LIN {X 0,Y 86.241,Z 1157.577,A -85,B 0,C 180,E1 5429.612,E2 5429.612} C_VEL
LIN {X 0,Y 83.784,Z 1172.301,A -85,B 0,C 180,E1 5420.249,E2 5420.249} C_VEL
LIN {X 0,Y 83.269,Z 1185.193,A -85,B 0,C 180,E1 5410.109,E2 5410.109} C_VEL
LIN {X 0,Y 85.244,Z 1197.586,A -85,B 0,C 180,E1 5398.656,E2 5398.656} C_VEL
LIN {X 0,Y 91.359,Z 1209.722,A -85,B 0,C 180,E1 5386.067,E2 5386.067} C_VEL
LIN {X 0,Y 101.878,Z 1220.023,A -85,B 0,C 180,E1 5375.037,E2 5375.037} C_VEL
LIN {X 0,Y 114.698,Z 1227.862,A -85,B 0,C 180,E1 5366.799,E2 5366.799} C_VEL
LIN {X 0,Y 97.634,Z 1225.464,A -85,B 0,C 180,E1 5353.315,E2 5353.315} C_VEL
LIN {X 0,Y 88.981,Z 1221.588,A -85,B 0,C 180,E1 5336.7,E2 5336.7} C_VEL
LIN {X 0,Y 88.107,Z 1220.31,A -85,B 0,C 180,E1 5331.809,E2 5331.809} C_VEL
LIN {X 0,Y 85.061,Z 1227.697,A -85,B 0,C 180,E1 5324.282,E2 5324.282} C_VEL
LIN {X 0,Y 85.385,Z 1239.016,A -85,B 0,C 180,E1 5311.333,E2 5311.333} C_VEL
LIN {X 0,Y 86.182,Z 1243.374,A -85,B 0,C 180,E1 5305.333,E2 5305.333} C_VEL
LIN {X 0,Y 85.817,Z 1248.62,A -85,B 0,C 180,E1 5294.447,E2 5294.447} C_VEL
LIN {X 0,Y 90.743,Z 1255.131,A -85,B 0,C 180,E1 5277.312,E2 5277.312} C_VEL
LIN {X 0,Y 102.644,Z 1259.967,A -85,B 0,C 180,E1 5263.088,E2 5263.088} C_VEL
LIN {X 0,Y 89.773,Z 1251.394,A -85,B 0,C 180,E1 5248.616,E2 5248.616} C_VEL
LIN {X 0,Y 84.154,Z 1242.377,A -85,B 0,C 180,E1 5233.747,E2 5233.747} C_VEL
LIN {X 0,Y 82.846,Z 1235.817,A -85,B 0,C 180,E1 5224.153,E2 5224.153} C_VEL
LIN {X 0,Y 82.358,Z 1227.952,A -85,B 0,C 180,E1 5214.426,E2 5214.426} C_VEL
LIN {X 0,Y 83.548,Z 1216.638,A -85,B 0,C 180,E1 5202.591,E2 5202.591} C_VEL
LIN {X 0,Y 87.163,Z 1203.687,A -85,B 0,C 180,E1 5191.683,E2 5191.683} C_VEL
LIN {X 0,Y 88.042,Z 1198.552,A -85,B 0,C 180,E1 5187.954,E2 5187.954} C_VEL
LIN {X 0,Y 88.162,Z 1183.445,A -85,B 0,C 180,E1 5178.16,E2 5178.16} C_VEL
LIN {X 0,Y 89.756,Z 1178.502,A -85,B 0,C 180,E1 5175.416,E2 5175.416} C_VEL
LIN {X 0,Y 98.668,Z 1160.656,A -85,B 0,C 180,E1 5167.456,E2 5167.456} C_VEL
LIN {X 0,Y 108.892,Z 1140.068,A -85,B 0,C 180,E1 5160.845,E2 5160.845} C_VEL
LIN {X 0,Y 119.307,Z 1117.626,A -85,B 0,C 180,E1 5155.718,E2 5155.718} C_VEL
LIN {X 0,Y 129.224,Z 1093.9,A -85,B 0,C 180,E1 5151.794,E2 5151.794} C_VEL
LIN {X 0,Y 137.935,Z 1070.062,A -85,B 0,C 180,E1 5148.915,E2 5148.915} C_VEL
LIN {X 0,Y 145.83,Z 1044.502,A -85,B 0,C 180,E1 5146.657,E2 5146.657} C_VEL
LIN {X 0,Y 152.519,Z 1017.799,A -85,B 0,C 180,E1 5144.946,E2 5144.946} C_VEL
LIN {X 0,Y 182.121,Z 883.493,A -85,B 0,C 180,E1 5138.791,E2 5138.791} C_VEL
LIN {X 0,Y 178.666,Z 874.642,A -85,B 0,C 180,E1 5136.269,E2 5136.269} C_VEL
LIN {X 0,Y 168.951,Z 876.076,A -85,B 0,C 180,E1 5132.04,E2 5132.04} C_VEL
LIN {X 0,Y 161.363,Z 878.264,A -85,B 0,C 180,E1 5128.389,E2 5128.389} C_VEL
LIN {X 0,Y 158.218,Z 879.25,A -85,B 0,C 180,E1 5126.744,E2 5126.744} C_VEL
LIN {X 0,Y 157.864,Z 879.467,A -85,B 0,C 180,E1 5126.374,E2 5126.374} C_VEL
LIN {X 0,Y 158.802,Z 887.342,A -85,B 0,C 180,E1 5122.407,E2 5122.407} C_VEL
LIN {X 0,Y 137.912,Z 929.195,A -85,B 0,C 180,E1 5115.445,E2 5115.445} C_VEL
LIN {X 0,Y 129.417,Z 947.663,A -85,B 0,C 180,E1 5111.944,E2 5111.944} C_VEL
LIN {X 0,Y 118.078,Z 998.542,A -85,B 0,C 180,E1 5108.011,E2 5108.011} C_VEL
LIN {X 0,Y 108.514,Z 1037.175,A -85,B 0,C 180,E1 5103.701,E2 5103.701} C_VEL
LIN {X 0,Y 99.397,Z 1074.485,A -85,B 0,C 180,E1 5097.673,E2 5097.673} C_VEL
LIN {X 0,Y 91.918,Z 1104.757,A -85,B 0,C 180,E1 5091.009,E2 5091.009} C_VEL
LIN {X 0,Y 86.721,Z 1124.357,A -85,B 0,C 180,E1 5085.162,E2 5085.162} C_VEL
LIN {X 0,Y 82.161,Z 1140.976,A -85,B 0,C 180,E1 5078.365,E2 5078.365} C_VEL
LIN {X 0,Y 78.202,Z 1157.109,A -85,B 0,C 180,E1 5069.627,E2 5069.627} C_VEL
LIN {X 0,Y 75.851,Z 1171.444,A -85,B 0,C 180,E1 5059.643,E2 5059.643} C_VEL
LIN {X 0,Y 75.568,Z 1184.592,A -85,B 0,C 180,E1 5048.369,E2 5048.369} C_VEL
LIN {X 0,Y 77.98,Z 1196.619,A -85,B 0,C 180,E1 5036.324,E2 5036.324} C_VEL
LIN {X 0,Y 84.068,Z 1207.905,A -85,B 0,C 180,E1 5024.124,E2 5024.124} C_VEL
LIN {X 0,Y 95.246,Z 1218.728,A -85,B 0,C 180,E1 5012.49,E2 5012.49} C_VEL
LIN {X 0,Y 104.27,Z 1224.54,A -85,B 0,C 180,E1 5006.526,E2 5006.526} C_VEL
LIN {X 0,Y 87.98,Z 1221.298,A -85,B 0,C 180,E1 4991.224,E2 4991.224} C_VEL
LIN {X 0,Y 81.108,Z 1216.92,A -85,B 0,C 180,E1 4973.223,E2 4973.223} C_VEL
LIN {X 0,Y 77.596,Z 1224.563,A -85,B 0,C 180,E1 4964.885,E2 4964.885} C_VEL
LIN {X 0,Y 77.861,Z 1236.114,A -85,B 0,C 180,E1 4950.726,E2 4950.726} C_VEL
LIN {X 0,Y 78.846,Z 1240.177,A -85,B 0,C 180,E1 4944.897,E2 4944.897} C_VEL
LIN {X 0,Y 78.56,Z 1244.991,A -85,B 0,C 180,E1 4934.487,E2 4934.487} C_VEL
LIN {X 0,Y 82.705,Z 1251.194,A -85,B 0,C 180,E1 4917.852,E2 4917.852} C_VEL
LIN {X 0,Y 93.414,Z 1256.211,A -85,B 0,C 180,E1 4903.24,E2 4903.24} C_VEL
LIN {X 0,Y 81.625,Z 1247.63,A -85,B 0,C 180,E1 4888.538,E2 4888.538} C_VEL
LIN {X 0,Y 76.334,Z 1238.553,A -85,B 0,C 180,E1 4872.867,E2 4872.867} C_VEL
LIN {X 0,Y 75.088,Z 1232.042,A -85,B 0,C 180,E1 4863.053,E2 4863.053} C_VEL
LIN {X 0,Y 74.723,Z 1222.958,A -85,B 0,C 180,E1 4851.536,E2 4851.536} C_VEL
LIN {X 0,Y 76.489,Z 1211.523,A -85,B 0,C 180,E1 4839.332,E2 4839.332} C_VEL
LIN {X 0,Y 81.228,Z 1197.323,A -85,B 0,C 180,E1 4827.206,E2 4827.206} C_VEL
LIN {X 0,Y 88.468,Z 1181.188,A -85,B 0,C 180,E1 4816.82,E2 4816.82} C_VEL
LIN {X 0,Y 89.756,Z 1178.502,A -85,B 0,C 180,E1 4815.416,E2 4815.416} C_VEL
LIN {X 0,Y 91.632,Z 1172.758,A -85,B 0,C 180,E1 4812.391,E2 4812.391} C_VEL
LIN {X 0,Y 94.055,Z 1156.183,A -85,B 0,C 180,E1 4804.217,E2 4804.217} C_VEL
LIN {X 0,Y 96.111,Z 1150.794,A -85,B 0,C 180,E1 4802.181,E2 4802.181} C_VEL
LIN {X 0,Y 106.915,Z 1129.286,A -85,B 0,C 180,E1 4796.127,E2 4796.127} C_VEL
LIN {X 0,Y 117.252,Z 1106.872,A -85,B 0,C 180,E1 4791.639,E2 4791.639} C_VEL
LIN {X 0,Y 126.869,Z 1083.26,A -85,B 0,C 180,E1 4788.25,E2 4788.25} C_VEL
LIN {X 0,Y 135.738,Z 1057.899,A -85,B 0,C 180,E1 4785.61,E2 4785.61} C_VEL
LIN {X 0,Y 143.195,Z 1032.145,A -85,B 0,C 180,E1 4783.666,E2 4783.666} C_VEL
LIN {X 0,Y 157.748,Z 968.792,A -85,B 0,C 180,E1 4780.37,E2 4780.37} C_VEL
LIN {X 0,Y 176.471,Z 886.212,A -85,B 0,C 180,E1 4776.883,E2 4776.883} C_VEL
LIN {X 0,Y 175.082,Z 882.618,A -85,B 0,C 180,E1 4775.801,E2 4775.801} C_VEL
LIN {X 0,Y 165.031,Z 884.421,A -85,B 0,C 180,E1 4771.383,E2 4771.383} C_VEL
LIN {X 0,Y 156.456,Z 887.466,A -85,B 0,C 180,E1 4767.166,E2 4767.166} C_VEL
LIN {X 0,Y 153.441,Z 888.778,A -85,B 0,C 180,E1 4765.52,E2 4765.52} C_VEL
LIN {X 0,Y 152.755,Z 888.903,A -85,B 0,C 180,E1 4765.03,E2 4765.03} C_VEL
LIN {X 0,Y 152.718,Z 890.398,A -85,B 0,C 180,E1 4764.383,E2 4764.383} C_VEL
LIN {X 0,Y 130.69,Z 933.07,A -85,B 0,C 180,E1 4757.287,E2 4757.287} C_VEL
LIN {X 0,Y 123.411,Z 948.435,A -85,B 0,C 180,E1 4754.382,E2 4754.382} C_VEL
LIN {X 0,Y 111.781,Z 998.605,A -85,B 0,C 180,E1 4750.492,E2 4750.492} C_VEL
LIN {X 0,Y 101.944,Z 1036.897,A -85,B 0,C 180,E1 4746.187,E2 4746.187} C_VEL
LIN {X 0,Y 93.403,Z 1069.952,A -85,B 0,C 180,E1 4740.747,E2 4740.747} C_VEL
LIN {X 0,Y 85.152,Z 1101.651,A -85,B 0,C 180,E1 4733.549,E2 4733.549} C_VEL
LIN {X 0,Y 80.078,Z 1120.078,A -85,B 0,C 180,E1 4727.983,E2 4727.983} C_VEL
LIN {X 0,Y 74.964,Z 1137.836,A -85,B 0,C 180,E1 4720.528,E2 4720.528} C_VEL
LIN {X 0,Y 70.694,Z 1154.219,A -85,B 0,C 180,E1 4711.208,E2 4711.208} C_VEL
LIN {X 0,Y 68.052,Z 1169.443,A -85,B 0,C 180,E1 4699.752,E2 4699.752} C_VEL
LIN {X 0,Y 67.837,Z 1182.497,A -85,B 0,C 180,E1 4687.623,E2 4687.623} C_VEL
LIN {X 0,Y 70.599,Z 1194.922,A -85,B 0,C 180,E1 4674.31,E2 4674.31} C_VEL
LIN {X 0,Y 77.394,Z 1206.485,A -85,B 0,C 180,E1 4661.156,E2 4661.156} C_VEL
LIN {X 0,Y 88.2,Z 1216.728,A -85,B 0,C 180,E1 4650.079,E2 4650.079} C_VEL
LIN {X 0,Y 93.813,Z 1220.694,A -85,B 0,C 180,E1 4645.948,E2 4645.948} C_VEL
LIN {X 0,Y 78.673,Z 1216.583,A -85,B 0,C 180,E1 4628.505,E2 4628.505} C_VEL
LIN {X 0,Y 74.391,Z 1213.178,A -85,B 0,C 180,E1 4615.037,E2 4615.037} C_VEL
LIN {X 0,Y 70.422,Z 1220.557,A -85,B 0,C 180,E1 4606.485,E2 4606.485} C_VEL
LIN {X 0,Y 70.379,Z 1233.071,A -85,B 0,C 180,E1 4589.989,E2 4589.989} C_VEL
LIN {X 0,Y 71.54,Z 1237.335,A -85,B 0,C 180,E1 4583.569,E2 4583.569} C_VEL
LIN {X 0,Y 71.81,Z 1243.099,A -85,B 0,C 180,E1 4569.618,E2 4569.618} C_VEL
LIN {X 0,Y 79.308,Z 1249.887,A -85,B 0,C 180,E1 4549.973,E2 4549.973} C_VEL
LIN {X 0,Y 84.334,Z 1252.112,A -85,B 0,C 180,E1 4543.446,E2 4543.446} C_VEL
LIN {X 0,Y 72.537,Z 1242.379,A -85,B 0,C 180,E1 4526.174,E2 4526.174} C_VEL
LIN {X 0,Y 68.592,Z 1234.322,A -85,B 0,C 180,E1 4511.776,E2 4511.776} C_VEL
LIN {X 0,Y 67.364,Z 1227.852,A -85,B 0,C 180,E1 4501.701,E2 4501.701} C_VEL
LIN {X 0,Y 67.195,Z 1218.248,A -85,B 0,C 180,E1 4488.846,E2 4488.846} C_VEL
LIN {X 0,Y 69.965,Z 1205.301,A -85,B 0,C 180,E1 4474.612,E2 4474.612} C_VEL
LIN {X 0,Y 76.007,Z 1190.131,A -85,B 0,C 180,E1 4461.808,E2 4461.808} C_VEL
LIN {X 0,Y 84.267,Z 1173.415,A -85,B 0,C 180,E1 4451.622,E2 4451.622} C_VEL
LIN {X 0,Y 94.036,Z 1154.74,A -85,B 0,C 180,E1 4443.577,E2 4443.577} C_VEL
LIN {X 0,Y 96.111,Z 1150.794,A -85,B 0,C 180,E1 4442.181,E2 4442.181} C_VEL
LIN {X 0,Y 98.404,Z 1144.528,A -85,B 0,C 180,E1 4439.954,E2 4439.954} C_VEL
LIN {X 0,Y 101.798,Z 1126.829,A -85,B 0,C 180,E1 4433.486,E2 4433.486} C_VEL
LIN {X 0,Y 104.003,Z 1121.008,A -85,B 0,C 180,E1 4431.976,E2 4431.976} C_VEL
LIN {X 0,Y 114.099,Z 1098.922,A -85,B 0,C 180,E1 4428.042,E2 4428.042} C_VEL
LIN {X 0,Y 123.604,Z 1075.322,A -85,B 0,C 180,E1 4425.009,E2 4425.009} C_VEL
LIN {X 0,Y 131.796,Z 1051.416,A -85,B 0,C 180,E1 4422.768,E2 4422.768} C_VEL
LIN {X 0,Y 139.117,Z 1025.432,A -85,B 0,C 180,E1 4421.017,E2 4421.017} C_VEL
LIN {X 0,Y 170.63,Z 890.747,A -85,B 0,C 180,E1 4414.994,E2 4414.994} C_VEL
LIN {X 0,Y 160.368,Z 893.274,A -85,B 0,C 180,E1 4410.362,E2 4410.362} C_VEL
LIN {X 0,Y 155.446,Z 895.26,A -85,B 0,C 180,E1 4407.959,E2 4407.959} C_VEL
LIN {X 0,Y 152.869,Z 896.535,A -85,B 0,C 180,E1 4406.63,E2 4406.63} C_VEL
LIN {X 0,Y 130.942,Z 939.04,A -85,B 0,C 180,E1 4399.93,E2 4399.93} C_VEL
LIN {X 0,Y 125.047,Z 951.051,A -85,B 0,C 180,E1 4397.83,E2 4397.83} C_VEL
LIN {X 0,Y 114.292,Z 981.442,A -85,B 0,C 180,E1 4395.905,E2 4395.905} C_VEL
LIN {X 0,Y 105.613,Z 1003.909,A -85,B 0,C 180,E1 4393.356,E2 4393.356} C_VEL
LIN {X 0,Y 102.058,Z 1012.732,A -85,B 0,C 180,E1 4391.867,E2 4391.867} C_VEL
LIN {X 0,Y 92.223,Z 1048.643,A -85,B 0,C 180,E1 4387.159,E2 4387.159} C_VEL
LIN {X 0,Y 82.48,Z 1084.483,A -85,B 0,C 180,E1 4380.088,E2 4380.088} C_VEL
LIN {X 0,Y 75.142,Z 1110.38,A -85,B 0,C 180,E1 4372.978,E2 4372.978} C_VEL
LIN {X 0,Y 69.631,Z 1128.783,A -85,B 0,C 180,E1 4365.889,E2 4365.889} C_VEL
LIN {X 0,Y 64.799,Z 1145.279,A -85,B 0,C 180,E1 4356.999,E2 4356.999} C_VEL
LIN {X 0,Y 61.007,Z 1161.901,A -85,B 0,C 180,E1 4344.705,E2 4344.705} C_VEL
LIN {X 0,Y 59.871,Z 1174.778,A -85,B 0,C 180,E1 4332.539,E2 4332.539} C_VEL
LIN {X 0,Y 61.526,Z 1187.718,A -85,B 0,C 180,E1 4318.137,E2 4318.137} C_VEL
LIN {X 0,Y 67.553,Z 1200.569,A -85,B 0,C 180,E1 4302.781,E2 4302.781} C_VEL
LIN {X 0,Y 77.41,Z 1211.28,A -85,B 0,C 180,E1 4290.604,E2 4290.604} C_VEL
LIN {X 0,Y 83.85,Z 1216.333,A -85,B 0,C 180,E1 4285.349,E2 4285.349} C_VEL
LIN {X 0,Y 69.97,Z 1211.478,A -85,B 0,C 180,E1 4265.457,E2 4265.457} C_VEL
LIN {X 0,Y 67.67,Z 1209.506,A -85,B 0,C 180,E1 4257.01,E2 4257.01} C_VEL
LIN {X 0,Y 63.147,Z 1217.105,A -85,B 0,C 180,E1 4247.495,E2 4247.495} C_VEL
LIN {X 0,Y 62.214,Z 1226.228,A -85,B 0,C 180,E1 4234.597,E2 4234.597} C_VEL
LIN {X 0,Y 64.298,Z 1234.06,A -85,B 0,C 180,E1 4222.392,E2 4222.392} C_VEL
LIN {X 0,Y 64.729,Z 1239.155,A -85,B 0,C 180,E1 4209.176,E2 4209.176} C_VEL
LIN {X 0,Y 71.354,Z 1245.628,A -85,B 0,C 180,E1 4189.851,E2 4189.851} C_VEL
LIN {X 0,Y 75.487,Z 1247.652,A -85,B 0,C 180,E1 4183.797,E2 4183.797} C_VEL
LIN {X 0,Y 64.209,Z 1237.526,A -85,B 0,C 180,E1 4164.863,E2 4164.863} C_VEL
LIN {X 0,Y 60.986,Z 1230.343,A -85,B 0,C 180,E1 4151.347,E2 4151.347} C_VEL
LIN {X 0,Y 59.619,Z 1223.429,A -85,B 0,C 180,E1 4140,E2 4140} C_VEL
LIN {X 0,Y 59.852,Z 1213.134,A -85,B 0,C 180,E1 4125.487,E2 4125.487} C_VEL
LIN {X 0,Y 63.655,Z 1199.427,A -85,B 0,C 180,E1 4109.783,E2 4109.783} C_VEL
LIN {X 0,Y 70.628,Z 1184.114,A -85,B 0,C 180,E1 4096.911,E2 4096.911} C_VEL
LIN {X 0,Y 80.2,Z 1166.199,A -85,B 0,C 180,E1 4086.471,E2 4086.471} C_VEL
LIN {X 0,Y 91.096,Z 1146.179,A -85,B 0,C 180,E1 4078.585,E2 4078.585} C_VEL
LIN {X 0,Y 102.412,Z 1124.236,A -85,B 0,C 180,E1 4072.684,E2 4072.684} C_VEL
LIN {X 0,Y 104.003,Z 1121.008,A -85,B 0,C 180,E1 4071.976,E2 4071.976} C_VEL
LIN {X 0,Y 106.407,Z 1114.29,A -85,B 0,C 180,E1 4070.312,E2 4070.312} C_VEL
LIN {X 0,Y 109.831,Z 1095.663,A -85,B 0,C 180,E1 4065.206,E2 4065.206} C_VEL
LIN {X 0,Y 111.823,Z 1089.589,A -85,B 0,C 180,E1 4064.146,E2 4064.146} C_VEL
LIN {X 0,Y 121.399,Z 1064.961,A -85,B 0,C 180,E1 4061.439,E2 4061.439} C_VEL
LIN {X 0,Y 129.737,Z 1039.244,A -85,B 0,C 180,E1 4059.422,E2 4059.422} C_VEL
LIN {X 0,Y 137.792,Z 1008.247,A -85,B 0,C 180,E1 4057.704,E2 4057.704} C_VEL
LIN {X 0,Y 163.71,Z 899.715,A -85,B 0,C 180,E1 4053.068,E2 4053.068} C_VEL
LIN {X 0,Y 155.007,Z 902.734,A -85,B 0,C 180,E1 4049.007,E2 4049.007} C_VEL
LIN {X 0,Y 154.109,Z 903.377,A -85,B 0,C 180,E1 4048.61,E2 4048.61} C_VEL
LIN {X 0,Y 131.432,Z 946.581,A -85,B 0,C 180,E1 4042.185,E2 4042.185} C_VEL
LIN {X 0,Y 127.866,Z 953.811,A -85,B 0,C 180,E1 4041.022,E2 4041.022} C_VEL
LIN {X 0,Y 116.923,Z 984.271,A -85,B 0,C 180,E1 4039.393,E2 4039.393} C_VEL
LIN {X 0,Y 107.983,Z 1006.831,A -85,B 0,C 180,E1 4037.145,E2 4037.145} C_VEL
LIN {X 0,Y 104.093,Z 1016.054,A -85,B 0,C 180,E1 4035.833,E2 4035.833} C_VEL
LIN {X 0,Y 95.358,Z 1038.552,A -85,B 0,C 180,E1 4033.626,E2 4033.626} C_VEL
LIN {X 0,Y 88.201,Z 1053.887,A -85,B 0,C 180,E1 4031.192,E2 4031.192} C_VEL
LIN {X 0,Y 82.755,Z 1063.928,A -85,B 0,C 180,E1 4028.491,E2 4028.491} C_VEL
LIN {X 0,Y 80.102,Z 1068.347,A -85,B 0,C 180,E1 4026.56,E2 4026.56} C_VEL
LIN {X 0,Y 71.181,Z 1098.56,A -85,B 0,C 180,E1 4018.968,E2 4018.968} C_VEL
LIN {X 0,Y 64.536,Z 1120.073,A -85,B 0,C 180,E1 4011.484,E2 4011.484} C_VEL
LIN {X 0,Y 58.856,Z 1137.813,A -85,B 0,C 180,E1 4002.303,E2 4002.303} C_VEL
LIN {X 0,Y 54.29,Z 1154.517,A -85,B 0,C 180,E1 3990.077,E2 3990.077} C_VEL
LIN {X 0,Y 52.178,Z 1170.174,A -85,B 0,C 180,E1 3974.426,E2 3974.426} C_VEL
LIN {X 0,Y 53.472,Z 1183.047,A -85,B 0,C 180,E1 3958.929,E2 3958.929} C_VEL
LIN {X 0,Y 59.626,Z 1196.715,A -85,B 0,C 180,E1 3941.421,E2 3941.421} C_VEL
LIN {X 0,Y 71.291,Z 1209.221,A -85,B 0,C 180,E1 3926.839,E2 3926.839} C_VEL
LIN {X 0,Y 74.077,Z 1211.506,A -85,B 0,C 180,E1 3924.52,E2 3924.52} C_VEL
LIN {X 0,Y 61.702,Z 1205.805,A -85,B 0,C 180,E1 3901.22,E2 3901.22} C_VEL
LIN {X 0,Y 61.262,Z 1205.553,A -85,B 0,C 180,E1 3899.57,E2 3899.57} C_VEL
LIN {X 0,Y 56.24,Z 1212.882,A -85,B 0,C 180,E1 3889.728,E2 3889.728} C_VEL
LIN {X 0,Y 54.697,Z 1222.858,A -85,B 0,C 180,E1 3874.179,E2 3874.179} C_VEL
LIN {X 0,Y 57.226,Z 1231.046,A -85,B 0,C 180,E1 3860.178,E2 3860.178} C_VEL
LIN {X 0,Y 59.262,Z 1237.624,A -85,B 0,C 180,E1 3840.691,E2 3840.691} C_VEL
LIN {X 0,Y 66.721,Z 1242.79,A -85,B 0,C 180,E1 3824.176,E2 3824.176} C_VEL
LIN {X 0,Y 56.233,Z 1232.772,A -85,B 0,C 180,E1 3804.14,E2 3804.14} C_VEL
LIN {X 0,Y 53.335,Z 1226.121,A -85,B 0,C 180,E1 3790.805,E2 3790.805} C_VEL
LIN {X 0,Y 51.837,Z 1218.002,A -85,B 0,C 180,E1 3776.683,E2 3776.683} C_VEL
LIN {X 0,Y 53.115,Z 1206.093,A -85,B 0,C 180,E1 3759.042,E2 3759.042} C_VEL
LIN {X 0,Y 58.731,Z 1191.339,A -85,B 0,C 180,E1 3742.2,E2 3742.2} C_VEL
LIN {X 0,Y 67.682,Z 1174.467,A -85,B 0,C 180,E1 3729.14,E2 3729.14} C_VEL
LIN {X 0,Y 78.312,Z 1155.916,A -85,B 0,C 180,E1 3719.746,E2 3719.746} C_VEL
LIN {X 0,Y 89.582,Z 1135.744,A -85,B 0,C 180,E1 3712.95,E2 3712.95} C_VEL
LIN {X 0,Y 101.06,Z 1113.322,A -85,B 0,C 180,E1 3707.869,E2 3707.869} C_VEL
LIN {X 0,Y 111.823,Z 1089.589,A -85,B 0,C 180,E1 3704.146,E2 3704.146} C_VEL
LIN {X 0,Y 114.015,Z 1082.548,A -85,B 0,C 180,E1 3702.929,E2 3702.929} C_VEL
LIN {X 0,Y 116.898,Z 1063.17,A -85,B 0,C 180,E1 3698.799,E2 3698.799} C_VEL
LIN {X 0,Y 118.559,Z 1056.901,A -85,B 0,C 180,E1 3698.022,E2 3698.022} C_VEL
LIN {X 0,Y 126.419,Z 1031.788,A -85,B 0,C 180,E1 3696.318,E2 3696.318} C_VEL
LIN {X 0,Y 143.061,Z 965.183,A -85,B 0,C 180,E1 3693.205,E2 3693.205} C_VEL
LIN {X 0,Y 156.818,Z 909.33,A -85,B 0,C 180,E1 3691.101,E2 3691.101} C_VEL
LIN {X 0,Y 155.742,Z 909.851,A -85,B 0,C 180,E1 3690.601,E2 3690.601} C_VEL
LIN {X 0,Y 131.238,Z 955.759,A -85,B 0,C 180,E1 3684.127,E2 3684.127} C_VEL
LIN {X 0,Y 119.951,Z 987.012,A -85,B 0,C 180,E1 3682.733,E2 3682.733} C_VEL
LIN {X 0,Y 110.678,Z 1009.923,A -85,B 0,C 180,E1 3680.75,E2 3680.75} C_VEL
LIN {X 0,Y 106.854,Z 1018.842,A -85,B 0,C 180,E1 3679.648,E2 3679.648} C_VEL
LIN {X 0,Y 97.685,Z 1041.502,A -85,B 0,C 180,E1 3677.831,E2 3677.831} C_VEL
LIN {X 0,Y 90.244,Z 1056.755,A -85,B 0,C 180,E1 3675.811,E2 3675.811} C_VEL
LIN {X 0,Y 84.295,Z 1067.126,A -85,B 0,C 180,E1 3673.47,E2 3673.47} C_VEL
LIN {X 0,Y 81.116,Z 1071.955,A -85,B 0,C 180,E1 3671.652,E2 3671.652} C_VEL
LIN {X 0,Y 73.032,Z 1086.127,A -85,B 0,C 180,E1 3668.592,E2 3668.592} C_VEL
LIN {X 0,Y 66.455,Z 1096.19,A -85,B 0,C 180,E1 3664.525,E2 3664.525} C_VEL
LIN {X 0,Y 63.262,Z 1100.726,A -85,B 0,C 180,E1 3661.308,E2 3661.308} C_VEL
LIN {X 0,Y 56.301,Z 1121.534,A -85,B 0,C 180,E1 3653.052,E2 3653.052} C_VEL
LIN {X 0,Y 50.344,Z 1139.22,A -85,B 0,C 180,E1 3642.476,E2 3642.476} C_VEL
LIN {X 0,Y 46.006,Z 1155.035,A -85,B 0,C 180,E1 3628.564,E2 3628.564} C_VEL
LIN {X 0,Y 44.501,Z 1170.405,A -85,B 0,C 180,E1 3610.355,E2 3610.355} C_VEL
LIN {X 0,Y 47.281,Z 1183.953,A -85,B 0,C 180,E1 3591.487,E2 3591.487} C_VEL
LIN {X 0,Y 54.446,Z 1196.027,A -85,B 0,C 180,E1 3575.014,E2 3575.014} C_VEL
LIN {X 0,Y 64.526,Z 1206.157,A -85,B 0,C 180,E1 3563.115,E2 3563.115} C_VEL
LIN {X 0,Y 55.09,Z 1201.442,A -85,B 0,C 180,E1 3542.664,E2 3542.664} C_VEL
LIN {X 0,Y 49.548,Z 1208.48,A -85,B 0,C 180,E1 3532.528,E2 3532.528} C_VEL
LIN {X 0,Y 47.15,Z 1217.89,A -85,B 0,C 180,E1 3516.07,E2 3516.07} C_VEL
LIN {X 0,Y 50.232,Z 1227.785,A -85,B 0,C 180,E1 3497.628,E2 3497.628} C_VEL
LIN {X 0,Y 54.099,Z 1235.084,A -85,B 0,C 180,E1 3473.723,E2 3473.723} C_VEL
LIN {X 0,Y 58.181,Z 1237.652,A -85,B 0,C 180,E1 3464.799,E2 3464.799} C_VEL
LIN {X 0,Y 48.935,Z 1228.594,A -85,B 0,C 180,E1 3445.41,E2 3445.41} C_VEL
LIN {X 0,Y 46.078,Z 1222.661,A -85,B 0,C 180,E1 3432.533,E2 3432.533} C_VEL
LIN {X 0,Y 44.326,Z 1214.897,A -85,B 0,C 180,E1 3417.414,E2 3417.414} C_VEL
LIN {X 0,Y 45.746,Z 1202.717,A -85,B 0,C 180,E1 3396.831,E2 3396.831} C_VEL
LIN {X 0,Y 52.288,Z 1187.401,A -85,B 0,C 180,E1 3377.987,E2 3377.987} C_VEL
LIN {X 0,Y 62.331,Z 1170,A -85,B 0,C 180,E1 3364.295,E2 3364.295} C_VEL
LIN {X 0,Y 73.905,Z 1150.91,A -85,B 0,C 180,E1 3354.978,E2 3354.978} C_VEL
LIN {X 0,Y 85.5,Z 1130.751,A -85,B 0,C 180,E1 3348.689,E2 3348.689} C_VEL
LIN {X 0,Y 97.369,Z 1107.93,A -85,B 0,C 180,E1 3343.966,E2 3343.966} C_VEL
LIN {X 0,Y 108.334,Z 1083.7,A -85,B 0,C 180,E1 3340.592,E2 3340.592} C_VEL
LIN {X 0,Y 117.933,Z 1058.751,A -85,B 0,C 180,E1 3338.165,E2 3338.165} C_VEL
LIN {X 0,Y 118.559,Z 1056.901,A -85,B 0,C 180,E1 3338.022,E2 3338.022} C_VEL
LIN {X 0,Y 120.376,Z 1049.693,A -85,B 0,C 180,E1 3337.152,E2 3337.152} C_VEL
LIN {X 0,Y 121.837,Z 1034.965,A -85,B 0,C 180,E1 3334.544,E2 3334.544} C_VEL
LIN {X 0,Y 122.826,Z 1026.483,A -85,B 0,C 180,E1 3333.335,E2 3333.335} C_VEL
LIN {X 0,Y 123.552,Z 1023.272,A -85,B 0,C 180,E1 3333.082,E2 3333.082} C_VEL
LIN {X 0,Y 144.608,Z 939.909,A -85,B 0,C 180,E1 3329.634,E2 3329.634} C_VEL
LIN {X 0,Y 134.291,Z 959.419,A -85,B 0,C 180,E1 3327.03,E2 3327.03} C_VEL
LIN {X 0,Y 123.297,Z 989.603,A -85,B 0,C 180,E1 3325.939,E2 3325.939} C_VEL
LIN {X 0,Y 113.819,Z 1012.796,A -85,B 0,C 180,E1 3324.208,E2 3324.208} C_VEL
LIN {X 0,Y 109.93,Z 1021.683,A -85,B 0,C 180,E1 3323.284,E2 3323.284} C_VEL
LIN {X 0,Y 100.989,Z 1043.278,A -85,B 0,C 180,E1 3321.931,E2 3321.931} C_VEL
LIN {X 0,Y 92.365,Z 1060.363,A -85,B 0,C 180,E1 3320.104,E2 3320.104} C_VEL
LIN {X 0,Y 85.406,Z 1071.744,A -85,B 0,C 180,E1 3317.844,E2 3317.844} C_VEL
LIN {X 0,Y 82.266,Z 1076.323,A -85,B 0,C 180,E1 3316.496,E2 3316.496} C_VEL
LIN {X 0,Y 73.4,Z 1090.843,A -85,B 0,C 180,E1 3313.82,E2 3313.82} C_VEL
LIN {X 0,Y 66.403,Z 1100.685,A -85,B 0,C 180,E1 3310.242,E2 3310.242} C_VEL
LIN {X 0,Y 62.752,Z 1105.337,A -85,B 0,C 180,E1 3307.544,E2 3307.544} C_VEL
LIN {X 0,Y 55.369,Z 1116.089,A -85,B 0,C 180,E1 3303.368,E2 3303.368} C_VEL
LIN {X 0,Y 49.619,Z 1124.021,A -85,B 0,C 180,E1 3297.818,E2 3297.818} C_VEL
LIN {X 0,Y 45.641,Z 1129.64,A -85,B 0,C 180,E1 3291.053,E2 3291.053} C_VEL
LIN {X 0,Y 39.779,Z 1147.02,A -85,B 0,C 180,E1 3276.208,E2 3276.208} C_VEL
LIN {X 0,Y 36.92,Z 1162.135,A -85,B 0,C 180,E1 3257.332,E2 3257.332} C_VEL
LIN {X 0,Y 38.663,Z 1177.043,A -85,B 0,C 180,E1 3234.062,E2 3234.062} C_VEL
LIN {X 0,Y 45.175,Z 1189.445,A -85,B 0,C 180,E1 3215.131,E2 3215.131} C_VEL
LIN {X 0,Y 55.395,Z 1200.42,A -85,B 0,C 180,E1 3201.418,E2 3201.418} C_VEL
LIN {X 0,Y 49.351,Z 1197.104,A -85,B 0,C 180,E1 3186.685,E2 3186.685} C_VEL
LIN {X 0,Y 42.656,Z 1204.661,A -85,B 0,C 180,E1 3174.936,E2 3174.936} C_VEL
LIN {X 0,Y 39.812,Z 1214.883,A -85,B 0,C 180,E1 3154.301,E2 3154.301} C_VEL
LIN {X 0,Y 43.456,Z 1224.452,A -85,B 0,C 180,E1 3133.954,E2 3133.954} C_VEL
LIN {X 0,Y 48.533,Z 1231.378,A -85,B 0,C 180,E1 3108.735,E2 3108.735} C_VEL
LIN {X 0,Y 49.717,Z 1232.143,A -85,B 0,C 180,E1 3105.56,E2 3105.56} C_VEL
LIN {X 0,Y 41.354,Z 1223.663,A -85,B 0,C 180,E1 3085.799,E2 3085.799} C_VEL
LIN {X 0,Y 38.362,Z 1217.844,A -85,B 0,C 180,E1 3072.035,E2 3072.035} C_VEL
LIN {X 0,Y 36.782,Z 1207.183,A -85,B 0,C 180,E1 3049.03,E2 3049.03} C_VEL
LIN {X 0,Y 40.624,Z 1193.838,A -85,B 0,C 180,E1 3025.521,E2 3025.521} C_VEL
LIN {X 0,Y 49.334,Z 1178.158,A -85,B 0,C 180,E1 3007.772,E2 3007.772} C_VEL
LIN {X 0,Y 61.415,Z 1159.289,A -85,B 0,C 180,E1 2995.366,E2 2995.366} C_VEL
LIN {X 0,Y 73.968,Z 1139.124,A -85,B 0,C 180,E1 2987.633,E2 2987.633} C_VEL
LIN {X 0,Y 86.032,Z 1117.929,A -85,B 0,C 180,E1 2982.505,E2 2982.505} C_VEL
LIN {X 0,Y 97.468,Z 1095.065,A -85,B 0,C 180,E1 2978.86,E2 2978.86} C_VEL
LIN {X 0,Y 107.635,Z 1071.558,A -85,B 0,C 180,E1 2976.283,E2 2976.283} C_VEL
LIN {X 0,Y 116.578,Z 1046.829,A -85,B 0,C 180,E1 2974.376,E2 2974.376} C_VEL
LIN {X 0,Y 123.552,Z 1023.272,A -85,B 0,C 180,E1 2973.082,E2 2973.082} C_VEL
LIN {X 0,Y 124.259,Z 1018.26,A -85,B 0,C 180,E1 2972.468,E2 2972.468} C_VEL
LIN {X 0,Y 123.856,Z 1005.172,A -85,B 0,C 180,E1 2969.625,E2 2969.625} C_VEL
LIN {X 0,Y 124.516,Z 1000.841,A -85,B 0,C 180,E1 2969.164,E2 2969.164} C_VEL
LIN {X 0,Y 126.198,Z 994.21,A -85,B 0,C 180,E1 2968.883,E2 2968.883} C_VEL
LIN {X 0,Y 116.611,Z 1017.122,A -85,B 0,C 180,E1 2967.364,E2 2967.364} C_VEL
LIN {X 0,Y 113.422,Z 1024.356,A -85,B 0,C 180,E1 2966.735,E2 2966.735} C_VEL
LIN {X 0,Y 104.77,Z 1044.81,A -85,B 0,C 180,E1 2965.802,E2 2965.802} C_VEL
LIN {X 0,Y 95.455,Z 1062.935,A -85,B 0,C 180,E1 2964.341,E2 2964.341} C_VEL
LIN {X 0,Y 87.758,Z 1075.115,A -85,B 0,C 180,E1 2962.42,E2 2962.42} C_VEL
LIN {X 0,Y 84.464,Z 1079.656,A -85,B 0,C 180,E1 2961.296,E2 2961.296} C_VEL
LIN {X 0,Y 75.304,Z 1094.013,A -85,B 0,C 180,E1 2959.291,E2 2959.291} C_VEL
LIN {X 0,Y 67.589,Z 1104.262,A -85,B 0,C 180,E1 2956.32,E2 2956.32} C_VEL
LIN {X 0,Y 63.461,Z 1109.176,A -85,B 0,C 180,E1 2953.97,E2 2953.97} C_VEL
LIN {X 0,Y 55.179,Z 1120.363,A -85,B 0,C 180,E1 2950.44,E2 2950.44} C_VEL
LIN {X 0,Y 48.387,Z 1128.552,A -85,B 0,C 180,E1 2945.401,E2 2945.401} C_VEL
LIN {X 0,Y 43.577,Z 1134.234,A -85,B 0,C 180,E1 2939.367,E2 2939.367} C_VEL
LIN {X 0,Y 35.147,Z 1145.667,A -85,B 0,C 180,E1 2927.703,E2 2927.703} C_VEL
LIN {X 0,Y 29.804,Z 1155.433,A -85,B 0,C 180,E1 2908.015,E2 2908.015} C_VEL
LIN {X 0,Y 29.293,Z 1159.117,A -85,B 0,C 180,E1 2897.2,E2 2897.2} C_VEL
LIN {X 0,Y 31.45,Z 1173.669,A -85,B 0,C 180,E1 2870.112,E2 2870.112} C_VEL
LIN {X 0,Y 39.621,Z 1186.982,A -85,B 0,C 180,E1 2847.997,E2 2847.997} C_VEL
LIN {X 0,Y 46.538,Z 1194.165,A -85,B 0,C 180,E1 2838.737,E2 2838.737} C_VEL
LIN {X 0,Y 43.819,Z 1192.711,A -85,B 0,C 180,E1 2831.408,E2 2831.408} C_VEL
LIN {X 0,Y 36.998,Z 1199.285,A -85,B 0,C 180,E1 2820.871,E2 2820.871} C_VEL
LIN {X 0,Y 32.551,Z 1208.917,A -85,B 0,C 180,E1 2798.811,E2 2798.811} C_VEL
LIN {X 0,Y 36.894,Z 1220.95,A -85,B 0,C 180,E1 2769.349,E2 2769.349} C_VEL
LIN {X 0,Y 41.474,Z 1226.362,A -85,B 0,C 180,E1 2746.836,E2 2746.836} C_VEL
LIN {X 0,Y 33.713,Z 1218.407,A -85,B 0,C 180,E1 2726.416,E2 2726.416} C_VEL
LIN {X 0,Y 29.879,Z 1210.496,A -85,B 0,C 180,E1 2705.762,E2 2705.762} C_VEL
LIN {X 0,Y 30.256,Z 1198.707,A -85,B 0,C 180,E1 2676.635,E2 2676.635} C_VEL
LIN {X 0,Y 37.753,Z 1183.587,A -85,B 0,C 180,E1 2650.898,E2 2650.898} C_VEL
LIN {X 0,Y 49.684,Z 1165.814,A -85,B 0,C 180,E1 2635.091,E2 2635.091} C_VEL
LIN {X 0,Y 62.453,Z 1146.835,A -85,B 0,C 180,E1 2626.134,E2 2626.134} C_VEL
LIN {X 0,Y 75.228,Z 1126.207,A -85,B 0,C 180,E1 2620.4,E2 2620.4} C_VEL
LIN {X 0,Y 87.549,Z 1103.669,A -85,B 0,C 180,E1 2616.471,E2 2616.471} C_VEL
LIN {X 0,Y 98.7,Z 1080.019,A -85,B 0,C 180,E1 2613.741,E2 2613.741} C_VEL
LIN {X 0,Y 108.541,Z 1055.139,A -85,B 0,C 180,E1 2611.781,E2 2611.781} C_VEL
LIN {X 0,Y 117.052,Z 1028.738,A -85,B 0,C 180,E1 2610.325,E2 2610.325} C_VEL
LIN {X 0,Y 124.516,Z 1000.841,A -85,B 0,C 180,E1 2609.164,E2 2609.164} C_VEL
LIN {X 0,Y 128.234,Z 1001.365,A -85,B 0,C 180,E1 2608.586,E2 2608.586} C_VEL
LIN {X 0,Y 128.234,Z 1082.056,A -85,B 0,C 180,E1 2608.586,E2 2608.586} C_VEL
LIN {X 0,Y 106.998,Z 1082.056,A -85,B 0,C 180,E1 2609.097,E2 2609.097} C_VEL
LIN {X 0,Y 105.001,Z 1080.056,A -85,B 0,C 180,E1 2609.156,E2 2609.156} C_VEL
LIN {X 0,Y 105.001,Z 1062.228,A -85,B 0,C 180,E1 2609.156,E2 2609.156} C_VEL
LIN {X 0,Y 101.411,Z 1061.174,A -85,B 0,C 180,E1 2608.66,E2 2608.66} C_VEL
LIN {X 0,Y 92.106,Z 1076.222,A -85,B 0,C 180,E1 2607.127,E2 2607.127} C_VEL
LIN {X 0,Y 86.723,Z 1083.65,A -85,B 0,C 180,E1 2605.812,E2 2605.812} C_VEL
LIN {X 0,Y 76.878,Z 1098.482,A -85,B 0,C 180,E1 2604.255,E2 2604.255} C_VEL
LIN {X 0,Y 68.684,Z 1108.673,A -85,B 0,C 180,E1 2601.868,E2 2601.868} C_VEL
LIN {X 0,Y 64.443,Z 1113.488,A -85,B 0,C 180,E1 2600.15,E2 2600.15} C_VEL
LIN {X 0,Y 55.328,Z 1124.938,A -85,B 0,C 180,E1 2597.395,E2 2597.395} C_VEL
LIN {X 0,Y 47.578,Z 1133.516,A -85,B 0,C 180,E1 2592.906,E2 2592.906} C_VEL
LIN {X 0,Y 42.943,Z 1138.127,A -85,B 0,C 180,E1 2588.649,E2 2588.649} C_VEL
LIN {X 0,Y 33.503,Z 1149.077,A -85,B 0,C 180,E1 2579.539,E2 2579.539} C_VEL
LIN {X 0,Y 25.864,Z 1158.83,A -85,B 0,C 180,E1 2561.089,E2 2561.089} C_VEL
LIN {X 0,Y 23.649,Z 1163.773,A -85,B 0,C 180,E1 2545.012,E2 2545.012} C_VEL
LIN {X 0,Y 24.541,Z 1177.106,A -85,B 0,C 180,E1 2503.429,E2 2503.429} C_VEL
LIN {X 0,Y 36.671,Z 1189.725,A -85,B 0,C 180,E1 2475.394,E2 2475.394} C_VEL
LIN {X 0,Y 28.401,Z 1197.938,A -85,B 0,C 180,E1 2459.499,E2 2459.499} C_VEL
LIN {X 0,Y 25.408,Z 1207.7,A -85,B 0,C 180,E1 2429.969,E2 2429.969} C_VEL
LIN {X 0,Y 30.905,Z 1217.439,A -85,B 0,C 180,E1 2401.995,E2 2401.995} C_VEL
LIN {X 0,Y 33.377,Z 1220.226,A -85,B 0,C 180,E1 2388.857,E2 2388.857} C_VEL
LIN {X 0,Y 27.432,Z 1214.498,A -85,B 0,C 180,E1 2373.145,E2 2373.145} C_VEL
LIN {X 0,Y 22.744,Z 1206.939,A -85,B 0,C 180,E1 2350.128,E2 2350.128} C_VEL
LIN {X 0,Y 23.472,Z 1194.014,A -85,B 0,C 180,E1 2309.257,E2 2309.257} C_VEL
LIN {X 0,Y 33.415,Z 1177.865,A -85,B 0,C 180,E1 2280.604,E2 2280.604} C_VEL
LIN {X 0,Y 46.934,Z 1159.53,A -85,B 0,C 180,E1 2266.525,E2 2266.525} C_VEL
LIN {X 0,Y 60.749,Z 1139.703,A -85,B 0,C 180,E1 2259.045,E2 2259.045} C_VEL
LIN {X 0,Y 73.727,Z 1118.808,A -85,B 0,C 180,E1 2254.569,E2 2254.569} C_VEL
LIN {X 0,Y 85.525,Z 1097.052,A -85,B 0,C 180,E1 2251.611,E2 2251.611} C_VEL
LIN {X 0,Y 96.892,Z 1072.352,A -85,B 0,C 180,E1 2249.417,E2 2249.417} C_VEL
LIN {X 0,Y 101.411,Z 1061.174,A -85,B 0,C 180,E1 2248.66,E2 2248.66} C_VEL
LIN {X 0,Y 105.102,Z 1061.943,A -85,B 0,C 180,E1 2248.059,E2 2248.059} C_VEL
LIN {X 0,Y 105.102,Z 1125.222,A -85,B 0,C 180,E1 2248.059,E2 2248.059} C_VEL
LIN {X 0,Y 79.854,Z 1125.222,A -85,B 0,C 180,E1 2248.955,E2 2248.955} C_VEL
LIN {X 0,Y 77.858,Z 1123.222,A -85,B 0,C 180,E1 2249.05,E2 2249.05} C_VEL
LIN {X 0,Y 77.858,Z 1109.57,A -85,B 0,C 180,E1 2249.05,E2 2249.05} C_VEL
LIN {X 0,Y 74.5,Z 1108.253,A -85,B 0,C 180,E1 2248.294,E2 2248.294} C_VEL
LIN {X 0,Y 66.64,Z 1116.932,A -85,B 0,C 180,E1 2246.198,E2 2246.198} C_VEL
LIN {X 0,Y 56.766,Z 1128.855,A -85,B 0,C 180,E1 2244.391,E2 2244.391} C_VEL
LIN {X 0,Y 48.554,Z 1137.277,A -85,B 0,C 180,E1 2241.3,E2 2241.3} C_VEL
LIN {X 0,Y 42.969,Z 1142.508,A -85,B 0,C 180,E1 2237.779,E2 2237.779} C_VEL
LIN {X 0,Y 31.812,Z 1154.027,A -85,B 0,C 180,E1 2230.551,E2 2230.551} C_VEL
LIN {X 0,Y 21.63,Z 1164.351,A -85,B 0,C 180,E1 2211.802,E2 2211.802} C_VEL
LIN {X 0,Y 18.49,Z 1168.61,A -85,B 0,C 180,E1 2196.502,E2 2196.502} C_VEL
LIN {X 0,Y 17.474,Z 1180.859,A -85,B 0,C 180,E1 2143.375,E2 2143.375} C_VEL
LIN {X 0,Y 25.925,Z 1189.872,A -85,B 0,C 180,E1 2115.48,E2 2115.48} C_VEL
LIN {X 0,Y 18.596,Z 1199.332,A -85,B 0,C 180,E1 2085.552,E2 2085.552} C_VEL
LIN {X 0,Y 21.83,Z 1209.904,A -85,B 0,C 180,E1 2042.7,E2 2042.7} C_VEL
LIN {X 0,Y 25.323,Z 1213.529,A -85,B 0,C 180,E1 2032.157,E2 2032.157} C_VEL
LIN {X 0,Y 19.09,Z 1207.671,A -85,B 0,C 180,E1 2015.18,E2 2015.18} C_VEL
LIN {X 0,Y 14.415,Z 1196.504,A -85,B 0,C 180,E1 1966.408,E2 1966.408} C_VEL
LIN {X 0,Y 22.905,Z 1181.231,A -85,B 0,C 180,E1 1919.179,E2 1919.179} C_VEL
LIN {X 0,Y 36.821,Z 1163.982,A -85,B 0,C 180,E1 1902.151,E2 1902.151} C_VEL
LIN {X 0,Y 50.673,Z 1145.684,A -85,B 0,C 180,E1 1894.813,E2 1894.813} C_VEL
LIN {X 0,Y 64.496,Z 1125.101,A -85,B 0,C 180,E1 1890.505,E2 1890.505} C_VEL
LIN {X 0,Y 74.5,Z 1108.253,A -85,B 0,C 180,E1 1888.294,E2 1888.294} C_VEL
LIN {X 0,Y 78.145,Z 1109.229,A -85,B 0,C 180,E1 1887.647,E2 1887.647} C_VEL
LIN {X 0,Y 78.145,Z 1160.358,A -85,B 0,C 180,E1 1887.647,E2 1887.647} C_VEL
LIN {X 0,Y 50.453,Z 1160.358,A -85,B 0,C 180,E1 1888.487,E2 1888.487} C_VEL
LIN {X 0,Y 48.455,Z 1158.358,A -85,B 0,C 180,E1 1888.585,E2 1888.585} C_VEL
LIN {X 0,Y 48.455,Z 1146.934,A -85,B 0,C 180,E1 1888.585,E2 1888.585} C_VEL
LIN {X 0,Y 45.464,Z 1145.327,A -85,B 0,C 180,E1 1887.23,E2 1887.23} C_VEL
LIN {X 0,Y 31.265,Z 1158.803,A -85,B 0,C 180,E1 1882.484,E2 1882.484} C_VEL
LIN {X 0,Y 19.266,Z 1168.926,A -85,B 0,C 180,E1 1869.097,E2 1869.097} C_VEL
LIN {X 0,Y 15.324,Z 1172.439,A -85,B 0,C 180,E1 1858.021,E2 1858.021} C_VEL
LIN {X 0,Y 11.402,Z 1186,A -85,B 0,C 180,E1 1773.992,E2 1773.992} C_VEL
LIN {X 0,Y 15.559,Z 1190.031,A -85,B 0,C 180,E1 1754.911,E2 1754.911} C_VEL
LIN {X 0,Y 11.755,Z 1200.031,A -85,B 0,C 180,E1 1695.148,E2 1695.148} C_VEL
LIN {X 0,Y 14.334,Z 1203.744,A -85,B 0,C 180,E1 1674.465,E2 1674.465} C_VEL
LIN {X 0,Y 7.268,Z 1191.82,A -85,B 0,C 180,E1 1595.625,E2 1595.625} C_VEL
LIN {X 0,Y 18.437,Z 1177.616,A -85,B 0,C 180,E1 1542.52,E2 1542.52} C_VEL
LIN {X 0,Y 34.001,Z 1159.879,A -85,B 0,C 180,E1 1530.97,E2 1530.97} C_VEL
LIN {X 0,Y 45.464,Z 1145.327,A -85,B 0,C 180,E1 1527.23,E2 1527.23} C_VEL
LIN {X 0,Y 48.937,Z 1146.535,A -85,B 0,C 180,E1 1526.104,E2 1526.104} C_VEL
LIN {X 0,Y 48.937,Z 1193.486,A -85,B 0,C 180,E1 1526.104,E2 1526.104} C_VEL
LIN {X 0,Y 14.366,Z 1193.486,A -85,B 0,C 180,E1 1524.346,E2 1524.346} C_VEL
LIN {X 0,Y 12.368,Z 1191.486,A -85,B 0,C 180,E1 1523.944,E2 1523.944} C_VEL
LIN {X 0,Y 12.368,Z 1182.307,A -85,B 0,C 180,E1 1523.944,E2 1523.944} C_VEL
LIN {X 0,Y 9.384,Z 1180.668,A -85,B 0,C 180,E1 1518.636,E2 1518.636} C_VEL
LIN {X 0,Y 5.326,Z 1190.327,A -85,B 0,C 180,E1 1388.768,E2 1388.768} C_VEL
LIN {X 0,Y 4.119,Z 1192.847,A -85,B 0,C 180,E1 1346.764,E2 1346.764} C_VEL
LIN {X 0,Y 9.384,Z 1180.668,A -85,B 0,C 180,E1 1518.636,E2 1518.636} C_VEL
LIN {X 0,Y 12.772,Z 1182.108,A -85,B 0,C 180,E1 1518.96,E2 1518.96} C_VEL
LIN {X 0,Y 12.772,Z 1317.5,A -85,B 0,C 180,E1 1518.96,E2 1518.96} C_VEL
LIN {X 0,Y 12.772,Z 1317.5,A -85,B 0,C 180,E1 1518.96,E2 1518.96}

QRS_NEXT_CUT()

QRS_NEXT()
QRS_HOME()

END
